FUNCTION_BLOCK FB_Sensor
VAR
	bDetect					AT %I* : BOOL;
END_VAR

PROPERTY Detect : BOOL
GET
Detect := bDetect;
END_GET
END_PROPERTY

END_FUNCTION_BLOCK

(* stored: Version 1.1.0.1, ProductVersion 3.1.4024.12
   POU FB_Sensor: Id {7ec15521-0f0e-4f12-94c5-2010fd0de13e}, SpecialFunc None
   Folder Properties: Id {56f5811e-5adc-4989-b537-50172fa88340}
   Property Detect: Id {c3635880-1a9c-40a8-b0d7-30611628ef17}
   Get Get: Id {eee2ea72-2eef-45ca-946e-39a6b9e92f97} *)
